# B&R Automation Studio project Tuerschleuse
Automation Studio 4.12.7.113

## Configuration Config1

CPU X20CP1584, AutomationRuntime J4.93, Build 4.1.2, Vc V4.73.2

### Task classes (Cpu.sw)
```
Cyclic#4:
  Program <- Program.prg
Libraries: standard
```

### Hardware
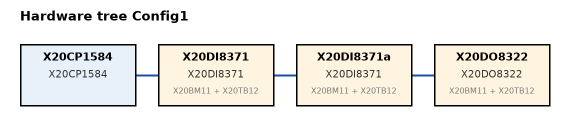
```
X20BM11 : X20BM11 v1.1.0.0  [X2X1 -> X20CP1584.IF6]
X20BM11a : X20BM11 v1.1.0.0  [X2X1 -> X20BM11.X2X2]
X20BM11b : X20BM11 v1.1.0.0  [X2X1 -> X20BM11a.X2X2]
X20CP1584 : X20CP1584 v1.10.0.0
  Connector IF2:
    ActivateDevice = 1
    Mode = Manual
    InternetAddress = 10.36.37.18
    SubnetMask = 255.250.255.0
  ConfigurationID = Tuerschleuse_Config1
  FileDevice1
  FileDeviceName1 = USER
  FileDevicePath1 = USER_PATH
X20DI8371 : X20DI8371 v1.4.0.0  [SS1 -> X20TB12.SS; SL -> X20BM11.SL1]
X20DI8371a : X20DI8371 v1.4.0.0  [SS1 -> X20TB12a.SS; SL -> X20BM11a.SL1]
X20DO8322 : X20DO8322 v1.5.0.0  [SS1 -> X20TB12b.SS; SL -> X20BM11b.SL1]
X20TB12 : X20TB12 v1.0.0.0
X20TB12a : X20TB12 v1.0.0.0
X20TB12b : X20TB12 v1.0.0.0
```

### IoMap.iom - X20CP1584/IoMap.iom
```iecst
VAR_CONFIG
	door_1.motor_closing AT %QX."X20DO8322".DigitalOutput01;
	door_1.motor_opening AT %QX."X20DO8322".DigitalOutput02;
	door_2.motor_opening AT %QX."X20DO8322".DigitalOutput03;
	door_2.motor_closing AT %QX."X20DO8322".DigitalOutput04;
	door_1.display AT %QX."X20DO8322".DigitalOutput05;
	door_2.display AT %QX."X20DO8322".DigitalOutput06;
	door_1.button_outside AT %IX."X20DI8371".DigitalInput01;
	door_2.button_outside AT %IX."X20DI8371".DigitalInput02;
	door_1.button_inside AT %IX."X20DI8371".DigitalInput03;
	door_2.button_inside AT %IX."X20DI8371".DigitalInput04;
	door_1.sensor_closed AT %IX."X20DI8371".DigitalInput05;
	door_1.sensor_opened AT %IX."X20DI8371".DigitalInput06;
	door_2.sensor_closed AT %IX."X20DI8371".DigitalInput07;
	door_2.sensor_opened AT %IX."X20DI8371".DigitalInput08;
	door_1.sensor_barrier AT %IX."X20DI8371a".DigitalInput01;
	door_2.sensor_barrier AT %IX."X20DI8371a".DigitalInput02;
END_VAR
```

## Logical view

### Global.typ
```iecst
TYPE
	door_t : 	STRUCT
		button_outside : BOOL;
		button_inside : BOOL;
		sensor_closed : BOOL;
		sensor_opened : BOOL;
		sensor_barrier : BOOL;
		motor_opening : BOOL;
		motor_closing : BOOL;
		display : BOOL;
		timer : TON;
	END_STRUCT;
END_TYPE
```

### Global.var
```iecst
VAR
	door_1 : door_t;
	door_2 : door_t;
END_VAR
```

### Program Logical/Program (ANSIC)

#### Cyclic.c - Cyclic code
```c
#include <bur/plctypes.h>

#ifdef _DEFAULT_INCLUDES
#include <AsDefault.h>
#endif

#include "state.h"
#include "door.h"
#include <stddef.h>

extern state_t* state;

void _CYCLIC ProgramCyclic(void)
{
	if (state != NULL)
	{
		state = state->run();
	}
	// TODO: error handling
}
```

#### Init.c - Initialization code
```c
#include <bur/plctypes.h>

#ifdef _DEFAULT_INCLUDES
#include <AsDefault.h>
#endif

#include "state.h"
#include "door.h"

state_t* state;
// door_t door_1;
// door_t door_2;

void _INIT ProgramInit(void)
{
	// set all output to zero
	door_1.motor_opening = FALSE;
	door_1.motor_closing = FALSE;
	door_1.display = FALSE;

	door_2.motor_opening = FALSE;
	door_2.motor_closing = FALSE;
	door_2.display = FALSE;

	// check for correct door position
	if (door_1.sensor_closed && door_2.sensor_closed)
	{
		// set state to DOORS_CLOSED
		state = &state_doors_closed;
	}
	else
	{
		state = &state_error;
	}
}
```

#### Exit.c - Exit code
```c
#include <bur/plctypes.h>

#ifdef _DEFAULT_INCLUDES
	#include <AsDefault.h>
#endif

#include "door.h"

// extern door_t door_1;
// extern door_t door_2;

void _EXIT ProgramExit(void)
{
	// set all output to zero
	door_1.motor_opening = FALSE;
	door_1.motor_closing = FALSE;
	door_1.display = FALSE;

	door_2.motor_opening = FALSE;
	door_2.motor_closing = FALSE;
	door_2.display = FALSE;
}
```

#### state.h
```c
#pragma once

#define DOOR_OPEN_TIMEOUT 5000 // 5 sec

typedef struct state* (*state_func_t)();
typedef struct state
{
	const char* name;
	state_func_t run;
} state_t;

extern state_t state_doors_closed;
extern state_t state_door_1_opening;
extern state_t state_door_2_opening;
extern state_t state_door_1_open;
extern state_t state_door_2_open;
extern state_t state_door_1_closing;
extern state_t state_door_2_closing;
extern state_t state_error;
```

#### state.c
```c
#include "state.h"
#include "door.h"
#include <stddef.h>

static state_t* state_func_doors_closed();
static state_t* state_func_door_1_opening();
static state_t* state_func_door_2_opening();
static state_t* state_func_door_1_open();
static state_t* state_func_door_2_open();
static state_t* state_func_door_1_closing();
static state_t* state_func_door_2_closing();
static state_t* state_func_error();

state_t state_doors_closed = 	{"Doors closed", state_func_doors_closed};
state_t state_door_1_opening = 	{"Door 1 opening", state_func_door_1_opening};
state_t state_door_2_opening = 	{"Door 2 opening", state_func_door_2_opening};
state_t state_door_1_open = 	{"Door 1 open", state_func_door_1_open};
state_t state_door_2_open = 	{"Door 2 open", state_func_door_2_open};
state_t state_door_1_closing = 	{"Door 1 closing", state_func_door_1_closing};
state_t state_door_2_closing = 	{"Door 2 closing", state_func_door_2_closing};
state_t state_error = 			{"Error", state_func_error};

// extern door_t door_1;
// extern door_t door_2;

state_t* state_func_doors_closed()
{
	if (door_1.button_outside || door_1.button_inside)
	{
		return &state_door_1_opening;
	}
	else if (door_2.button_outside || door_2.button_inside)
	{
		return &state_door_2_opening;
	}

	return &state_doors_closed;
}

state_t* state_func_door_1_opening()
{
	if (!door_1.motor_opening) door_1.motor_opening = TRUE;
	if (door_1.sensor_opened)
	{
		door_1.motor_opening = FALSE;
		// Fix? reset timer
		door_1.timer = set_TON(door_1.timer, FALSE, DOOR_OPEN_TIMEOUT);
		return &state_door_1_open;
	}
	// TODO: error handling
	return &state_door_1_opening;
}

state_t* state_func_door_1_open()
{
	door_1.timer = set_TON(door_1.timer, TRUE, DOOR_OPEN_TIMEOUT);
	if (door_1.timer.Q && door_1.sensor_barrier)
	{
		//door_1.timer = set_TON(door_1.timer, FALSE, DOOR_OPEN_TIMEOUT); // reset timer
		return &state_door_1_closing;
	}
	// TODO: error handling
	return &state_door_1_open;
}

state_t* state_func_door_1_closing()
{
	if (!door_1.motor_closing) door_1.motor_closing = TRUE;

	door_display(&door_1, BLINK_SLOW);

	if (!door_1.sensor_barrier || door_1.button_outside || door_1.button_inside)
	{
		door_1.motor_closing = FALSE;
		door_1.display = FALSE;
		return &state_door_1_opening;
	}
	else if (door_1.sensor_closed)
	{
		door_1.motor_closing = FALSE;
		door_1.display = FALSE;
		return &state_doors_closed;
	}
	// TODO: error handling
	return &state_door_1_closing;
}

state_t* state_func_door_2_opening()
{
	if (!door_2.motor_opening) door_2.motor_opening = TRUE;
	if (door_2.sensor_opened)
	{
		door_2.motor_opening = FALSE;
		// Fix? reset timer
		door_2.timer = set_TON(door_2.timer, FALSE, DOOR_OPEN_TIMEOUT);
		return &state_door_2_open;
	}
	// TODO: error handling
	return &state_door_2_opening;
}

state_t* state_func_door_2_open()
{
	door_2.timer = set_TON(door_2.timer, TRUE, DOOR_OPEN_TIMEOUT);
	if (door_2.timer.Q && door_2.sensor_barrier)
	{
		door_2.timer = set_TON(door_2.timer, FALSE, DOOR_OPEN_TIMEOUT); // reset timer
		return &state_door_2_closing;
	}
	// TODO: error handling
	return &state_door_2_open;
}

state_t* state_func_door_2_closing()
{
	if (!door_2.motor_closing) door_2.motor_closing = TRUE;

	door_display(&door_2, BLINK_SLOW);

	if (!door_2.sensor_barrier || door_2.button_outside || door_2.button_inside)
	{
		door_2.motor_closing = FALSE;
		door_2.display = FALSE;
		return &state_door_2_opening;
	}
	else if (door_2.sensor_closed)
	{
		door_2.motor_closing = FALSE;
		door_2.display = FALSE;
		return &state_doors_closed;
	}
	// TODO: error handling
	return &state_door_2_closing;
}

state_t* state_func_error()
{
	// TODO
	return &state_error;
}
```

#### door.h
```c
#pragma once

#include <bur/plctypes.h>

#ifdef _DEFAULT_INCLUDES
#include <AsDefault.h>
#endif

#define FALSE 0
#define TRUE  1
#define BLINK_SLOW	600
#define BLINK_FAST	200

/*
typedef struct door
{
	// inputs
	BOOL button_outside;
	BOOL button_inside;
	BOOL sensor_closed;
	BOOL sensor_opened;
	BOOL sensor_barrier;

	// outputs
	BOOL motor_opening;
	BOOL motor_closing;
	BOOL display;

	// intern
	TON_typ timer;
} door_t;
*/

void door_display(door_t* self, TIME blink_speed);
TON_typ set_TON(TON_typ TONset, BOOL in, TIME delay);
```

#### door.c
```c
#include "door.h"

void door_display(door_t* self, TIME blink_speed)
{
	self->timer.IN = TRUE;

	if (self->timer.Q)
	{
		self->display = !(self->display);
		self->timer.IN = FALSE;
	}

	self->timer = set_TON(self->timer, self->timer.IN, blink_speed);
}

TON_typ set_TON(TON_typ TONset, BOOL in, TIME delay)
{
	TONset.IN = in;
	TONset.PT = delay;
	TON(&TONset);
	return TONset;
}
```

Listed in the project but not available here: Logical/Program/Types.typ, Logical/Program/Variables.var
